(* IEC 61131-3 sources: plcassist-cli/packages/volt-lsp-iec/test-corpus/pro2193/Device/Plc Logic/Application/99 Library/Functions, 16 files *)

(* ---- DWORD_TO_HEXSTRING.fun ---- *)
// Convert PLC memory address into a string with hex characters represented by 0..9 and A..F.
FUNCTION DWORD_TO_HEXSTRING : STRING(8)
VAR_INPUT
	IN		: DWORD;		// Address - result of ADR()
END_VAR
VAR
	i		: USINT;
	temp	: BYTE;
	pt		: POINTER TO BYTE;
END_VAR

(*

Copy from oscat_basic_334 library

version 1.3	29. mar. 2008
programmer	hugo
tested by	tobias

DWORD_TO_STRINGH converts a DWORD to a String of Hexadecimal represented by '0' .. '9' and 'A' .. 'F'.
The lowest order Character will be on the right and the high order Character on the left.

*)

pt	:= ADR(DWORD_TO_HEXSTRING) + 8;					// Read output adress to pointer
pt^	:= 0;											// Write the closing byte (terminator) for the string

FOR i := 1 TO 8 DO									// Write the 8 hex characters backwards
	pt		:= pt - 1;								// Decrement the pointer
	temp	:= TO_BYTE(IN AND 16#0000000F);			// Read the lowest order hex value
	IF temp <= 9 THEN
		pt^	:= enumASCII.NUMBER_0 + temp;			// Convert value to hex character 0 - 9
	ELSE
		pt^	:= enumASCII.UPPERCASE_A + temp - 10;	// Convert value to hex character A - F
	END_IF
	IN		:= SHR(IN, 4);							// Shift 4 bits to right for next hex character
END_FOR

END_FUNCTION

(* ---- GetProjectInfo.fun ---- *)
// Reads the 'application info'. Rightclick on Application, Select Properties, Go to Information tab.
{attribute 'hide_all_locals'}
FUNCTION GetProjectInfo : ProjectInfoType
VAR_INPUT
END_VAR
VAR
	pApp		: POINTER TO CmpApp.APPLICATION;
	pAppInfo	: POINTER TO CmpApp.APPLICATION_INFO;
	iecResult	: SysTypes.RTS_IEC_RESULT;
END_VAR

// Get handle to current PLC application
pApp		:= CmpApp.AppGetCurrent(pResult := ADR(iecResult));
IF pApp = 0 THEN
	GetProjectInfo.projectName	:= 'ERROR READING CURRENT APP';
	RETURN;
END_IF

pAppInfo	:= CmpApp.AppGetApplicationInfo(pApp := pApp, pResult := ADR(iecResult));
IF pAppInfo = 0 THEN
	GetProjectInfo.projectName	:= 'ERROR GETTING APPLICATION INFO';
	RETURN;
END_IF

GetProjectInfo.projectName		:= pAppInfo^.pstProjectName^;
GetProjectInfo.author			:= pAppInfo^.pstAuthor^;
GetProjectInfo.version			:= pAppInfo^.pstVersion^;
GetProjectInfo.description		:= pAppInfo^.pstDescription^;
GetProjectInfo.profile			:= pAppInfo^.pstProfile^;
GetProjectInfo.lastChanges		:= DT_TO_STRING(pAppInfo^.dtLastChanges);

IF GetProjectInfo.projectName = '' THEN
	GetProjectInfo.projectName	:= 'INVALID PROJECTNAME';
END_IF
IF LEN(GetProjectInfo.lastChanges) > 3 THEN
	GetProjectInfo.lastChanges	:= RIGHT(GetProjectInfo.lastChanges, LEN(GetProjectInfo.lastChanges) - 3);
END_IF

END_FUNCTION

(* ---- ParseInstanceName.fun ---- *)
FUNCTION ParseInstanceName
VAR_INPUT
	pInstanceName				: Stu.CharBufferPtr;	// Pointer to string(80)
END_VAR
VAR
	tempString					: STRING(80);
	i							: INT;
END_VAR
VAR CONSTANT
	dotString					: STRING(1) := '.';
	underscoreString			: STRING(1) := '_';
END_VAR

// Check if input string is not empty
IF Stu.StrIsNullOrEmptyA(pInstanceName) THEN
	RETURN;
END_IF

// Check if the input string starts with a known prefix
FOR i := 1 TO 5 DO
	CASE i OF
		1: tempString := 'Device.Application.';
		2: tempString := 'PLC.Application.';
		3: tempString := 'Device.Sim.Device.Application.';
		4: tempString := 'PLC.Sim.PLC.Application.';
		5: tempString := '';
	END_CASE

	IF Stu.StrCmpStartA(pString := pInstanceName, pPrefix := ADR(tempString)) = 0 THEN
		EXIT;
	END_IF
END_FOR

// If prefix is found, remove this prefix
IF i <> 5 THEN
	Stu.StrMidA(
		pst					:= pInstanceName,
		uiInputBufferSize	:= 80,
		iLength				:= TO_INT(StrLenA(pInstanceName) - StrLenA(ADR(tempString))),
		iPosition			:= TO_INT(StrLenA(ADR(tempString)) + 1),
		pstResult			:= pInstanceName,
		uiResultBufferSize	:= 80);
END_IF

// Find all '.' chars and replace with underscores
i := 1;		// Start search at position 1
WHILE (i := StrFindA(pst1 := pInstanceName, pst2 := ADR(dotString), uiSearchStart := TO_UINT(i))) > 0 DO
	StrReplaceA(
		pstInput			:= pInstanceName,
		uiInputBufferSize	:= 80,
		pstReplaceWith		:= ADR(underscoreString),
		iLengthInput		:= 1,	// Don't know function of this parameter..
		iLengthToReplace	:= 1,
		iLengthToReplaceWith:= 1,
		iPosition			:= i);	// i is position where the dot was found
END_WHILE

END_FUNCTION

(* ---- RANGE_TO_RANGE.fun ---- *)
// Used for mapping a real input value from one range to another.
FUNCTION RANGE_TO_RANGE : REAL
VAR_INPUT
	input		: REAL;	// input is limited to: input_LO <= input <= input_HI
	input_LO	: REAL;
	input_HI	: REAL;
	output_LO	: REAL;
	output_HI	: REAL;
END_VAR
VAR
	inputRange	: REAL;
	outputRange	: REAL;
END_VAR

(*

Zie hier voor voorbeeld:
https://stackoverflow.com/questions/929103/convert-a-number-range-to-another-range-maintaining-ratio

Update 24-03-2023: Added logic from SCALE_R function in Oscat library.
*)

inputRange	:= input_HI - input_LO;
outputRange	:= output_HI - output_LO;

IF inputRange = 0 THEN // Never divide by zero
	RANGE_TO_RANGE := output_LO;
ELSE
	RANGE_TO_RANGE := outputRange / inputRange * (LIMIT(input_LO, input, input_HI) - input_LO) + output_LO;
END_IF

END_FUNCTION

(* ---- RANGE_TO_WORD.fun ---- *)
// Used for mapping a REAL input value into a WORD (from 0 to 65535)
FUNCTION RANGE_TO_WORD : WORD
VAR_INPUT
	input		: REAL;	// input is limited to: input_LO <= input <= input_HI
	input_LO	: REAL;
	input_HI	: REAL;
END_VAR

// Update 24-03-2023: Added logic from RANGE_TO_WORD function in Oscat library.
// Update 08-06-2023: Removed logic here and use RANGE_TO_RANGE method instead (because devide by zero exception was possible)

RANGE_TO_WORD := TO_WORD(
					TRUNC(
						RANGE_TO_RANGE(
							input		:= input,
							input_LO	:= input_LO,
							input_HI	:= input_HI,
							output_LO	:= 0.0,
//							output_HI	:= 65535.0)));
							output_HI	:= 16384.0)));		// For Lenze analog outputs the maximum range is 16384.

// Example use:
// MapAnalogOut			:= Brink.RANGE_TO_WORD(input := rSetPointCharger,			input_LO := 0.0,	input_HI := rMaxChargerSetting);
// MapAnalogOut			:= Brink.RANGE_TO_WORD(input := profile.rVel,				input_LO := 0.0,	input_HI := rMaxSpeedSetting);
// wSetPointCharger		:= Brink.RANGE_TO_WORD(input := Data.rSetPointCharger,		input_LO := 0.0,	input_HI := 20.0);
// wSetPointCharger[i]	:= Brink.RANGE_TO_WORD(input := Data.rSetPointCharger[i],	input_LO := 0.0,	input_HI := 20.0);

END_FUNCTION

(* ---- Round.fun ---- *)
// This function rounds a real down to n digits behind the comma.
FUNCTION Round : REAL
VAR_INPUT
	in	: REAL;
	N	: USINT(0..4);
END_VAR
VAR
	X	: REAL;
END_VAR

(*
version 1.5	25. oct. 2008
programmer	hugo
tested by	tobias

this function rounds a real down to n digits behind the comma.

*)

CASE N OF
	0:	X := 1.0;
	1:	X := 10.0;
	2:	X := 100.0;
	3:	X := 1000.0;
	4:	X := 10000.0;
END_CASE

Round := TO_REAL(TO_DINT(in * X)) / X;

(* revision history
hm	1. sep 2006	rev 1.0
	original version

hm	2. dec 2007	rev 1.1
	changed code for better performance

hm	8. jan 2008	rev 1.2
	further improvement in performance

hm 11. mar. 2008	rev 1.3
	corrected an error with negative numbers
	use real_to_dint instead of trunc

hm	16. mar 2008	rev 1.4
	added type conversion to avoid warning under codesys 3.0

hm	25. oct. 2008	rev 1.5
	new code using global constants decades
*)

END_FUNCTION

(* ---- TaskDisableWatchdog.fun ---- *)
// Disable watchdog for the current task
// The watchdog is disabled only for the current cycle! At the next cycle, the watchod is automatically enabled!
FUNCTION TaskDisableWatchdog : BOOL
VAR
	iecResult		: SysTypes.RTS_IEC_RESULT;
	handle			: SysTypes.RTS_IEC_HANDLE;
END_VAR

handle				:= CmpIecTask.IecTaskGetCurrent(ADR(iecResult));			// Function to get own task handle

IF handle = SysTypes.RTS_INVALID_HANDLE THEN RETURN; END_IF
IF iecResult <> CmpErrors.Errors.ERR_OK THEN RETURN; END_IF

iecResult			:= CmpIecTask.IecTaskDisableWatchdog(hIecTask := handle);

IF iecResult <> CmpErrors.Errors.ERR_OK THEN RETURN; END_IF

TaskDisableWatchdog	:= TRUE;

END_FUNCTION

(* ---- TaskGetInfo.fun ---- *)
// Returns task interval value (in ms) of current task
// Do not call function each PLC cycle. Calling it once is enough.
FUNCTION TaskGetInfo : CmpIecTask.Task_Info2
VAR
	iecResult		: SysTypes.RTS_IEC_RESULT;
	handle			: SysTypes.RTS_IEC_HANDLE;
	pIecTaskInfo	: POINTER TO CmpIecTask.Task_Info2;
END_VAR

handle				:= CmpIecTask.IecTaskGetCurrent(ADR(iecResult));			// Function to get own task handle

IF handle = SysTypes.RTS_INVALID_HANDLE THEN RETURN; END_IF
IF iecResult <> CmpErrors.Errors.ERR_OK THEN RETURN; END_IF

pIecTaskInfo		:= CmpIecTask.IecTaskGetInfo3(hIecTask := handle, pResult := ADR(iecResult));	// Function returns the task information of the specified task

IF pIecTaskInfo = 0 THEN RETURN; END_IF

TaskGetInfo			:= pIecTaskInfo^;

END_FUNCTION

(* ---- TaskGetInterval.fun ---- *)
// Returns task interval value (in ms) of current task
// Do not call function each PLC cycle. Calling it once is enough.
FUNCTION TaskGetInterval : TIME
VAR_OUTPUT
	taskName		: STRING;
END_VAR
VAR
	iecResult		: SysTypes.RTS_IEC_RESULT;
	handle			: SysTypes.RTS_IEC_HANDLE;
	pIecTaskInfo	: POINTER TO CmpIecTask.Task_Info2;
END_VAR

handle				:= CmpIecTask.IecTaskGetCurrent(ADR(iecResult));			// Function to get own task handle

IF handle = SysTypes.RTS_INVALID_HANDLE THEN RETURN; END_IF
IF iecResult <> CmpErrors.Errors.ERR_OK THEN RETURN; END_IF

pIecTaskInfo		:= CmpIecTask.IecTaskGetInfo3(hIecTask := handle, pResult := ADR(iecResult));	// Function returns the task information of the specified task

IF pIecTaskInfo = 0 THEN RETURN; END_IF

taskName			:= pIecTaskInfo^.pszName^;
TaskGetInterval		:= TO_TIME(pIecTaskInfo^.dwInterval / 1000);

END_FUNCTION

(* ---- ThrowException.fun ---- *)
FUNCTION ThrowException : BOOL
VAR_INPUT
	message			: STRING := '';	// A custom message (reason of throwing the exception) to echo to the PLC log
END_VAR

LogPlc.Fatal(message);		// Add a custom message to the PLC log
LogPlc.Throw();

END_FUNCTION

(* ---- Arrays.prg ---- *)
// Helper functions for arrays
{attribute 'no_explicit_call' := 'Static helper class to do stuff with all kinds of arrays'}
{attribute 'hide_all_locals'}
PROGRAM Arrays

// Because arrays are value-type, it's not possible to cast an array of fbs to another type.
// More info here:
// https://stackoverflow.com/questions/69319659/how-do-i-pass-an-array-of-an-extended-type-in-codesys-twincat3

// The function Vacuum_ResetAll should not be needed !!!
// The interface IVacuum extends IActuator,
// so you should be able to use ActuatorResetAll for vacuums too
// However, this does not work with dynamic arrays
// You get error message: Cannot convert type 'ARRAY[1..3] of IVacuum' to type 'ARRAY[*] of IActuator
// Hopefully CODESYS fixes this in the future.

END_PROGRAM

// Returns true if all elements in the actuator array are equal to condition.
METHOD PUBLIC Actuator_All : BOOL
VAR_IN_OUT
	actuatorArray		: ARRAY[*] OF IActuator;
END_VAR
VAR_INPUT
	condition			: BOOL;
END_VAR
VAR
	upper, lower, di	: DINT;
END_VAR
%FOLDER Tests
lower	:= LOWER_BOUND(actuatorArray, 1);
upper	:= UPPER_BOUND(actuatorArray, 1);

Actuator_All := TRUE;

FOR di := lower TO upper DO
	IF actuatorArray[di] = 0 THEN
		LogPlc.Fatal('Actuator_All: Element in array of interfaces is NULL!');
		Actuator_All := FALSE;
		EXIT;
	ELSIF actuatorArray[di].Map() <> condition THEN
		Actuator_All := FALSE;
		EXIT;	// Exit the loop on the first match
	END_IF
END_FOR
END_METHOD

// Returns true if any element in the actuator array is equal to condition.
METHOD PUBLIC Actuator_Any : BOOL
VAR_IN_OUT
	actuatorArray		: ARRAY[*] OF IActuator;
END_VAR
VAR_INPUT
	condition			: BOOL;
END_VAR
VAR
	upper, lower, di	: DINT;
END_VAR
%FOLDER Tests
lower	:= LOWER_BOUND(actuatorArray, 1);
upper	:= UPPER_BOUND(actuatorArray, 1);

FOR di := lower TO upper DO
	IF actuatorArray[di] = 0 THEN
		LogPlc.Fatal('Actuator_Any: Element in array of interfaces is NULL!');
	ELSIF actuatorArray[di].Map() = condition THEN
		Actuator_Any := TRUE;
		EXIT;	// Exit the loop on the first match
	END_IF
END_FOR
END_METHOD

// Fires the Reset method on the actuator array
METHOD PUBLIC Actuator_ResetAll
VAR_IN_OUT
	actuatorArray		: ARRAY[*] OF IActuator;
END_VAR
VAR
	upper, lower, di	: DINT;
END_VAR
%FOLDER Execute methods
lower	:= LOWER_BOUND(actuatorArray, 1);
upper	:= UPPER_BOUND(actuatorArray, 1);

FOR di := lower TO upper DO
	IF actuatorArray[di] = 0 THEN
		LogPlc.Fatal('Actuator_ResetAll: Element in array of interfaces is NULL!');
	ELSE
		actuatorArray[di].Reset();
	END_IF
END_FOR
END_METHOD

// Returns true if all the modules (Xi, Xu, or Y unit) are in a safe position
METHOD PUBLIC AllUnitsAreInSafePosition : BOOL
VAR_IN_OUT
	safeModules			: ARRAY[*] OF IModuleHasSafePos;
END_VAR
VAR
	upper, lower, di	: DINT;
END_VAR
%FOLDER Tests
lower	:= LOWER_BOUND(safeModules, 1);
upper	:= UPPER_BOUND(safeModules, 1);

AllUnitsAreInSafePosition := TRUE;

FOR di := lower TO upper DO
	IF safeModules[di] = 0 THEN
		ThrowException('AllUnitsAreInSafePosition: Element in array of interfaces is NULL!');
	ELSIF NOT safeModules[di].InSafePos THEN
		AllUnitsAreInSafePosition := FALSE;
		EXIT;	// Exit the loop on the first match
	END_IF
END_FOR
END_METHOD

// Returns true if all elements in the bool array are equal to condition
METHOD PUBLIC Bool_All : BOOL
VAR_IN_OUT
	boolArray			: ARRAY[*] OF BOOL;
END_VAR
VAR_INPUT
	condition			: BOOL;
END_VAR
VAR
	upper, lower, di	: DINT;
END_VAR
%FOLDER Tests
lower	:= LOWER_BOUND(boolArray, 1);
upper	:= UPPER_BOUND(boolArray, 1);

Bool_All := TRUE;

FOR di := lower TO upper DO
	IF boolArray[di] <> condition THEN
		Bool_All := FALSE;
		EXIT;						// Exit the loop on the first match
	END_IF
END_FOR
END_METHOD

// Returns true if any element in the bool array is equal to condition
METHOD PUBLIC Bool_Any : BOOL
VAR_IN_OUT
	boolArray			: ARRAY[*] OF BOOL;
END_VAR
VAR_INPUT
	condition			: BOOL;
END_VAR
VAR
	upper, lower, di	: DINT;
END_VAR
%FOLDER Tests
lower	:= LOWER_BOUND(boolArray, 1);
upper	:= UPPER_BOUND(boolArray, 1);

FOR di := lower TO upper DO
	IF boolArray[di] = condition THEN
		Bool_Any := TRUE;
		EXIT;						// Exit the loop on the first match
	END_IF
END_FOR
END_METHOD

// Resets all booleans in an array
METHOD PUBLIC Bool_Reset
VAR_IN_OUT
	boolArray		: ARRAY[*] OF BOOL;
END_VAR
VAR
	upper, lower, di	: DINT;
END_VAR
%FOLDER Execute methods
lower	:= LOWER_BOUND(boolArray, 1);
upper	:= UPPER_BOUND(boolArray, 1);

FOR di := lower TO upper DO
	boolArray[di] := FALSE;
END_FOR
END_METHOD

// Sets all booleans in an array
METHOD PUBLIC Bool_Set
VAR_IN_OUT
	boolArray		: ARRAY[*] OF BOOL;
END_VAR
VAR
	upper, lower, di	: DINT;
END_VAR
%FOLDER Execute methods
lower	:= LOWER_BOUND(boolArray, 1);
upper	:= UPPER_BOUND(boolArray, 1);

FOR di := lower TO upper DO
	boolArray[di] := TRUE;
END_FOR
END_METHOD

// Returns true if all digital sensors in the array are equal to condition
METHOD PUBLIC DigitalSensor_All : BOOL
VAR_IN_OUT
	sensorArray			: ARRAY[*] OF DigitalSensorFB;
END_VAR
VAR_INPUT
	condition			: BOOL;		// TRUE = IsActive, FALSE = IsInactive
END_VAR
VAR
	upper, lower, di	: DINT;
END_VAR
%FOLDER Digital Sensors
lower	:= LOWER_BOUND(sensorArray, 1);
upper	:= UPPER_BOUND(sensorArray, 1);

DigitalSensor_All := TRUE;

FOR di := lower TO upper DO
	IF (condition AND NOT sensorArray[di].IsActive)
	OR (NOT condition AND NOT sensorArray[di].IsInactive)
	THEN
		DigitalSensor_All := FALSE;
		EXIT;						// Exit the loop on the first match
	END_IF
END_FOR
END_METHOD

// Returns true if any element in the bool array is equal to condition
METHOD PUBLIC DigitalSensor_Any : BOOL
VAR_IN_OUT
	sensorArray			: ARRAY[*] OF DigitalSensorFB;
END_VAR
VAR_INPUT
	condition			: BOOL;
END_VAR
VAR
	upper, lower, di	: DINT;
END_VAR
%FOLDER Digital Sensors
lower	:= LOWER_BOUND(sensorArray, 1);
upper	:= UPPER_BOUND(sensorArray, 1);

FOR di := lower TO upper DO
	IF (condition AND sensorArray[di].IsActive)
	OR (NOT condition AND sensorArray[di].IsInactive)
	THEN
		DigitalSensor_Any := TRUE;
		EXIT;						// Exit the loop on the first match
	END_IF
END_FOR
END_METHOD

// Returns true if all digital sensors (that are enabled) in the array are equal to condition
METHOD PUBLIC DigitalSensor_Enabled_All : BOOL
VAR_IN_OUT
	sensorArray			: ARRAY[*] OF DigitalSensorWithEnableFB;
END_VAR
VAR_INPUT
	bitMask				: DWORD;	// Only test sensors when corresponding bitnumber is high.
	condition			: BOOL;
END_VAR
VAR
	upper, lower, di	: DINT;
	counter				: USINT := 0;
END_VAR
%FOLDER Digital Sensors
lower	:= LOWER_BOUND(sensorArray, 1);
upper	:= UPPER_BOUND(sensorArray, 1);

DigitalSensor_Enabled_All := TRUE;

FOR di := lower TO upper DO

	IF NOT BitLogic.Extract(bitMask, counter) THEN	// not cavity disabled
		IF (condition AND NOT sensorArray[di].IsActive)
		OR (NOT condition AND NOT sensorArray[di].IsInactive)
		THEN
			IF sensorArray[di].IsEnabled THEN		//Only reset when sensor is enabled
				DigitalSensor_Enabled_All := FALSE;
				EXIT;						// Exit the loop on the first match
			END_IF
		END_IF
	END_IF

	Increment.AnyInt(counter);
END_FOR
END_METHOD

// Returns true if any element (that is enabled) in the bool array is equal to condition
METHOD PUBLIC DigitalSensor_Enabled_Any : BOOL
VAR_IN_OUT
	sensorArray			: ARRAY[*] OF DigitalSensorWithEnableFB;
END_VAR
VAR_INPUT
	bitMask				: DWORD;	// Only test sensors when corresponding bitnumber is high.
	condition			: BOOL;
END_VAR
VAR
	upper, lower, di	: DINT;
	counter				: USINT := 0;
END_VAR
%FOLDER Digital Sensors
lower	:= LOWER_BOUND(sensorArray, 1);
upper	:= UPPER_BOUND(sensorArray, 1);

FOR di := lower TO upper DO

	IF NOT BitLogic.Extract(bitMask, counter) THEN	// not cavity disabled
		IF (condition AND sensorArray[di].IsActive)
		OR (NOT condition AND sensorArray[di].IsInactive)
		THEN
			IF sensorArray[di].IsEnabled THEN		// Only set when sensor is enabled
				DigitalSensor_Enabled_Any := TRUE;
				EXIT;						// Exit the loop on the first match
			END_IF
		END_IF
	END_IF

	Increment.AnyInt(counter);
END_FOR
END_METHOD

// Returns the largest position in an array
METHOD PUBLIC Position_Largest : REAL
VAR_IN_OUT
	positionArray		: ARRAY[*] OF PositionWithProfileType;
END_VAR
VAR
	upper, lower, di	: DINT;
END_VAR
%FOLDER Positions
lower					:= LOWER_BOUND(positionArray, 1);
upper					:= UPPER_BOUND(positionArray, 1);
Position_Largest		:= GVL_Constants.RealSmallest;

FOR di := lower TO upper DO
	Position_Largest	:= MAX(positionArray[di].Pos.value, Position_Largest);
END_FOR
END_METHOD

// Returns the smallest position in an array
METHOD PUBLIC Position_Smallest : REAL
VAR_IN_OUT
	positionArray		: ARRAY[*] OF PositionWithProfileType;
END_VAR
VAR
	upper, lower, di	: DINT;
END_VAR
%FOLDER Positions
lower					:= LOWER_BOUND(positionArray, 1);
upper					:= UPPER_BOUND(positionArray, 1);
Position_Smallest		:= GVL_Constants.RealLargest;

FOR di := lower TO upper DO
	Position_Smallest	:= MIN(positionArray[di].Pos.value, Position_Smallest);
END_FOR
END_METHOD

// Returns true if all elements in the vacuum array are equal to condition. Option to test either vacuum high input, or vacuum set output.
METHOD PUBLIC Vacuum_All : BOOL
VAR_IN_OUT
	vacuumArray			: ARRAY[*] OF IVacuum;
END_VAR
VAR_INPUT
	condition			: BOOL;
	channel				: enumSelectIQ := enumSelectIQ.Output;	// Optional: Select to check the vacuum high input, the set output, or both
END_VAR
VAR
	upper, lower, di	: DINT;
END_VAR
%FOLDER Tests
lower	:= LOWER_BOUND(vacuumArray, 1);
upper	:= UPPER_BOUND(vacuumArray, 1);

Vacuum_All := TRUE;

FOR di := lower TO upper DO
	IF vacuumArray[di] = 0 THEN
		LogPlc.Fatal('Vacuum_All: Element in array of interfaces is NULL!');
		Vacuum_All := FALSE;
		EXIT;	// Exit the loop on the first match
	END_IF

	IF vacuumArray[di].IsHigh <> condition AND (channel = enumSelectIQ.Input OR channel = enumSelectIQ.Both)
	OR vacuumArray[di].IsTurnedOn <> condition AND (channel = enumSelectIQ.Output OR channel = enumSelectIQ.Both)
	THEN
		Vacuum_All := FALSE;
		EXIT;	// Exit the loop on the first match
	END_IF
END_FOR
END_METHOD

// Returns true if any element in the vacuum array is equal to condition. Option to test either vacuum high input, or vacuum set output.
METHOD PUBLIC Vacuum_Any : BOOL
VAR_IN_OUT
	vacuumArray			: ARRAY[*] OF IVacuum;
END_VAR
VAR_INPUT
	condition			: BOOL;
	channel				: enumSelectIQ := enumSelectIQ.Output;	// Optional: Select to check the vacuum high input, the set output, or both
END_VAR
VAR
	upper, lower, di	: DINT;
END_VAR
%FOLDER Tests
lower	:= LOWER_BOUND(vacuumArray, 1);
upper	:= UPPER_BOUND(vacuumArray, 1);

FOR di := lower TO upper DO
	IF vacuumArray[di] = 0 THEN
		LogPlc.Fatal('Vacuum_Any: Element in array of interfaces is NULL!');
		CONTINUE;
	END_IF
	CASE channel OF
		enumSelectIQ.Input:
			IF vacuumArray[di].IsHigh = condition THEN
				Vacuum_Any := TRUE;
				EXIT;	// Exit the loop on the first match
			END_IF
		enumSelectIQ.Output:
			IF vacuumArray[di].IsTurnedOn = condition THEN
				Vacuum_Any := TRUE;
				EXIT;	// Exit the loop on the first match
			END_IF
		enumSelectIQ.Both:
			IF vacuumArray[di].IsHigh = condition OR vacuumArray[di].IsTurnedOn = condition THEN
				Vacuum_Any := TRUE;
				EXIT;	// Exit the loop on the first match
			END_IF
	END_CASE
END_FOR
END_METHOD

// Returns true if all elements in the vacuum array (that are enabled) are equal to condition. Option to test either vacuum high input, or vacuum set output.
METHOD PUBLIC Vacuum_Enabled_All : BOOL
VAR_IN_OUT
	vacuumArray			: ARRAY[*] OF IVacuum;
END_VAR
VAR_INPUT
	bitMask				: WORD;	// Only test vacuums when corresponding bitnumber is high.
	condition			: BOOL;
	channel				: enumSelectIQ := enumSelectIQ.Output;	// Optional: Select to check the vacuum high input, the set output, or both
END_VAR
VAR
	upper, lower, di	: DINT;
END_VAR
%FOLDER Tests
lower	:= LOWER_BOUND(vacuumArray, 1);
upper	:= UPPER_BOUND(vacuumArray, 1);

Vacuum_Enabled_All := TRUE;

FOR di := lower TO upper DO
	IF vacuumArray[di] = 0 THEN
		LogPlc.Fatal('Vacuum_All: Element in array of interfaces is NULL!');
		Vacuum_Enabled_All := FALSE;
		EXIT;	// Exit the loop on the first match
	END_IF

	IF NOT BitLogic.Extract(bitMask, TO_USINT(di)) THEN
		CONTINUE;
	END_IF

	IF vacuumArray[di].IsHigh <> condition AND (channel = enumSelectIQ.Input OR channel = enumSelectIQ.Both)
	OR vacuumArray[di].IsTurnedOn <> condition AND (channel = enumSelectIQ.Output OR channel = enumSelectIQ.Both)
	THEN
		Vacuum_Enabled_All := FALSE;
		EXIT;	// Exit the loop on the first match
	END_IF
END_FOR
END_METHOD

// Returns true if any element in the vacuum array (that is enabled) is equal to condition. Option to test either vacuum high input, or vacuum set output.
METHOD PUBLIC Vacuum_Enabled_Any : BOOL
VAR_IN_OUT
	vacuumArray			: ARRAY[*] OF IVacuum;
END_VAR
VAR_INPUT
	bitMask				: WORD;	// Only test vacuums when corresponding bitnumber is high.
	condition			: BOOL;
	channel				: enumSelectIQ := enumSelectIQ.Output;	// Optional: Select to check the vacuum high input, the set output, or both
END_VAR
VAR
	upper, lower, di	: DINT;
END_VAR
%FOLDER Tests
lower	:= LOWER_BOUND(vacuumArray, 1);
upper	:= UPPER_BOUND(vacuumArray, 1);

FOR di := lower TO upper DO
	IF vacuumArray[di] = 0 THEN
		LogPlc.Fatal('Vacuum_Any: Element in array of interfaces is NULL!');
		CONTINUE;
	END_IF

	IF NOT BitLogic.Extract(bitMask, TO_USINT(di)) THEN
		CONTINUE;
	END_IF

	CASE channel OF
		enumSelectIQ.Input:
			IF vacuumArray[di].IsHigh = condition THEN
				Vacuum_Enabled_Any := TRUE;
				EXIT;	// Exit the loop on the first match
			END_IF
		enumSelectIQ.Output:
			IF vacuumArray[di].IsTurnedOn = condition THEN
				Vacuum_Enabled_Any := TRUE;
				EXIT;	// Exit the loop on the first match
			END_IF
		enumSelectIQ.Both:
			IF vacuumArray[di].IsHigh = condition OR vacuumArray[di].IsTurnedOn = condition THEN
				Vacuum_Enabled_Any := TRUE;
				EXIT;	// Exit the loop on the first match
			END_IF
	END_CASE
END_FOR
END_METHOD

// Fires the Release method on all elements in the vacuum array
METHOD PUBLIC Vacuum_ReleaseAll : BOOL
VAR_IN_OUT
	vacuumArray			: ARRAY[*] OF IVacuum;
END_VAR
VAR
	upper, lower, di	: DINT;
END_VAR
%FOLDER Execute methods
lower	:= LOWER_BOUND(vacuumArray, 1);
upper	:= UPPER_BOUND(vacuumArray, 1);

Vacuum_ReleaseAll := TRUE;

FOR di := lower TO upper DO
	IF vacuumArray[di] = 0 THEN
		LogPlc.Fatal('Vacuum_ReleaseAll: Element in array of interfaces is NULL!');
		Vacuum_ReleaseAll := FALSE;
	ELSIF NOT vacuumArray[di].Release() THEN
		Vacuum_ReleaseAll := FALSE;
	END_IF
END_FOR
END_METHOD

// Fires the Release method on some elements in the vacuum array. Only reset vacuums whose corresponding bit is high in the bitMask
// !Remember! Vacuum arrays usually start from 1. So to set the first vacuum, use the second bit (bitMask.1) in the bitMask!
METHOD PUBLIC Vacuum_ReleaseSelected : BOOL
VAR_IN_OUT
	vacuumArray			: ARRAY[*] OF IVacuum;
END_VAR
VAR_INPUT
	bitMask				: WORD;	// Release vacuum if corresponding bitnumber is high.
END_VAR
VAR
	upper, lower, di	: DINT;
END_VAR
%FOLDER Execute methods
lower	:= LOWER_BOUND(vacuumArray, 1);
upper	:= UPPER_BOUND(vacuumArray, 1);

Vacuum_ReleaseSelected := TRUE;

FOR di := lower TO upper DO
	IF BitLogic.Extract(bitMask, TO_USINT(di)) THEN
		IF vacuumArray[di] = 0 THEN
			LogPlc.Fatal('Vacuum_ReleaseSelected: Element in array of interfaces is NULL!');
			Vacuum_ReleaseSelected := FALSE;
		ELSIF NOT vacuumArray[di].Release() THEN
			Vacuum_ReleaseSelected := FALSE;
		END_IF
	END_IF
END_FOR

// Method will fail if upper limit of vacuum array > 16
END_METHOD

// Resets the vacuum suction cups that no longer have a product. Returns 0 if all suction cups are turned off.
METHOD PUBLIC Vacuum_ResetIfNotHigh : UINT
VAR_IN_OUT
	vacuumArray			: ARRAY[*] OF IVacuum;
END_VAR
VAR
	result				: UINT;
	upper, lower, di	: DINT;
END_VAR
%FOLDER Execute methods
lower	:= LOWER_BOUND(vacuumArray, 1);
upper	:= UPPER_BOUND(vacuumArray, 1);

FOR di := lower TO upper DO
	IF vacuumArray[di] = 0 THEN
		LogPlc.Fatal('Vacuum_ResetIfNotHigh: Element in array of interfaces is NULL!');
	ELSIF vacuumArray[di].IsHigh THEN
		BitLogic.Load(result, TRUE, TO_USINT(LIMIT(0, di, 15)));
	ELSE
		vacuumArray[di].Reset();
	END_IF
END_FOR

Vacuum_ResetIfNotHigh := result;
END_METHOD

// Returns true if some elements in the vacuum array are equal to condition.
// Only test vacuums whose corresponding bit is high in the bitMask
// Option to test either vacuum high input, or vacuum set output.
// !Remember! Vacuum arrays usually start from 1. So to set the first vacuum, use the second bit (bitMask.1) in the bitMask!
METHOD PUBLIC Vacuum_Selected : BOOL
VAR_IN_OUT
	vacuumArray			: ARRAY[*] OF IVacuum;
END_VAR
VAR_INPUT
	bitMask				: WORD;	// Test vacuum if corresponding bitnumber is high.
	condition			: BOOL;
	channel				: enumSelectIQ := enumSelectIQ.Output;	// Optional: Select to check the vacuum high input, the set output, or both
END_VAR
VAR
	upper, lower, di	: DINT;
END_VAR
%FOLDER Tests
lower	:= LOWER_BOUND(vacuumArray, 1);
upper	:= UPPER_BOUND(vacuumArray, 1);

Vacuum_Selected := TRUE;

FOR di := lower TO upper DO
	IF BitLogic.Extract(bitMask, TO_USINT(di)) THEN
		IF vacuumArray[di] = 0 THEN
			LogPlc.Fatal('Vacuum_Selected: Element in array of interfaces is NULL!');
			Vacuum_Selected := FALSE;
			EXIT;
		END_IF
		CASE channel OF
			enumSelectIQ.Input:
				IF vacuumArray[di].IsHigh <> condition THEN
					Vacuum_Selected := FALSE;
					EXIT;	// Exit the loop on the first match
				END_IF
			enumSelectIQ.Output:
				IF vacuumArray[di].IsTurnedOn <> condition THEN
					Vacuum_Selected := FALSE;
					EXIT;	// Exit the loop on the first match
				END_IF
			enumSelectIQ.Both:
				IF vacuumArray[di].IsHigh <> condition OR vacuumArray[di].IsTurnedOn <> condition THEN
					Vacuum_Selected := FALSE;
					EXIT;	// Exit the loop on the first match
				END_IF
		END_CASE
	END_IF
END_FOR

// Method will fail if upper limit of vacuum array > 16
END_METHOD

// Fires the Set method on all elements in the vacuum array. Return true if all vacuums are high.
METHOD PUBLIC Vacuum_SetAll : BOOL
VAR_IN_OUT
	vacuumArray			: ARRAY[*] OF IVacuum;
END_VAR
VAR
	upper, lower, di	: DINT;
END_VAR
%FOLDER Execute methods
lower	:= LOWER_BOUND(vacuumArray, 1);
upper	:= UPPER_BOUND(vacuumArray, 1);

Vacuum_SetAll := TRUE;

FOR di := lower TO upper DO
	IF vacuumArray[di] = 0 THEN
		LogPlc.Fatal('Vacuum_SetAll: Element in array of interfaces is NULL!');
		Vacuum_SetAll := FALSE;
	ELSIF NOT vacuumArray[di].Set() THEN
		Vacuum_SetAll := FALSE;
	END_IF
END_FOR
END_METHOD

// Fires the Set method on some elements in the vacuum array. Only set vacuums whose corresponding bit is high in the bitMask
// !Remember! Vacuum arrays usually start from 1. So to set the first vacuum, use the second bit (bitMask.1) in the bitMask!
METHOD PUBLIC Vacuum_SetSelected : BOOL
VAR_IN_OUT
	vacuumArray			: ARRAY[*] OF IVacuum;
END_VAR
VAR_INPUT
	bitMask				: WORD;	// Set vacuum if corresponding bitnumber is high.
END_VAR
VAR
	upper, lower, di	: DINT;
END_VAR
%FOLDER Execute methods
lower	:= LOWER_BOUND(vacuumArray, 1);
upper	:= UPPER_BOUND(vacuumArray, 1);

Vacuum_SetSelected := TRUE;

FOR di := lower TO upper DO
	IF BitLogic.Extract(bitMask, TO_USINT(di)) THEN
		IF vacuumArray[di] = 0 THEN
			LogPlc.Fatal('Vacuum_SetSelected: Element in array of interfaces is NULL!');
			Vacuum_SetSelected := FALSE;
		ELSIF NOT vacuumArray[di].Set() THEN
			Vacuum_SetSelected := FALSE;
		END_IF
	END_IF
END_FOR

// Method will fail if upper limit of vacuum array > 16
END_METHOD

(* ---- BitLogic.prg ---- *)
// Helper functions to set or reset bits in integers
{attribute 'no_explicit_call' := 'Static helper class to do various operations on bits in integers'}
{attribute 'hide_all_locals'}
PROGRAM BitLogic
VAR
	uInput		: PointerSizesUnion;
END_VAR

END_PROGRAM

// Population count: Count the number of bits that are 1 in a byte
METHOD PUBLIC CountByte : USINT
VAR_INPUT
	in	: BYTE;			// Count number of 1's
END_VAR

// This method uses Brian Kernighan's algorithm. Google it for more info.
WHILE in <> 0 DO
	in			:= in AND (in - 1);		// Subtracting 1 from a number flips all the bits after the rightmost set bit, including the rightmost set bit itself
	CountByte	:= CountByte + 1;
END_WHILE
END_METHOD

// Population count: Count the number of bits that are 1 in a dword
METHOD PUBLIC CountDWord : USINT
VAR_INPUT
	in	: DWORD;		// Count number of 1's
END_VAR

// This method uses Brian Kernighan's algorithm. Google it for more info.
WHILE in <> 0 DO
	in			:= in AND (in - 1);
	CountDWord	:= CountDWord + 1;
END_WHILE
END_METHOD

// Population count: Count the number of bits that are 1 in a word
METHOD PUBLIC CountWord : USINT
VAR_INPUT
	in	: WORD;			// Count number of 1's
END_VAR

// This method uses Brian Kernighan's algorithm. Google it for more info.
WHILE in <> 0 DO
	in			:= in AND (in - 1);
	CountWord	:= CountWord + 1;
END_WHILE
END_METHOD

// Extract a single bit from any integer type (usefull in FOR loops)
METHOD PUBLIC Extract : BOOL
VAR_INPUT
	in	: ANY_INT;		// extract bit from this integer
	N	: USINT(0..63);	// position of bit on the nth position from right (right is lowest bit)
END_VAR
ValidateInput(in.diSize, N);

uInput.p1_Byte := in.pValue;

CASE in.diSize OF
	1:	Extract := (SHR(uInput.p1_Byte^,	N) AND 16#00000001) > 0;
	2:	Extract := (SHR(uInput.p2_Word^,	N) AND 16#00000001) > 0;
	4:	Extract := (SHR(uInput.p4_DWord^,	N) AND 16#00000001) > 0;
	8:	Extract := (SHR(uInput.p8_LWord^,	N) AND 16#00000001) > 0;
END_CASE
END_METHOD

// Extract a single bit from a byte type (usefull in FOR loops)
METHOD PUBLIC ExtractFromByte : BOOL
VAR_INPUT
	in	: REFERENCE TO BYTE;	// extract bit from this byte
	N	: BYTE(0..7);			// position of bit on the nth position from right (right is lowest bit)
END_VAR

// This is a separate method from Extract(), because ANY_INT cannot be a reference.
ExtractFromByte := (SHR(in,	N) AND 16#00000001) > 0;
END_METHOD

// Extract a single bit from a DWORD type (usefull in FOR loops)
METHOD PUBLIC ExtractFromDWord : BOOL
VAR_INPUT
	in	: REFERENCE TO DWORD;	// extract bit from this byte
	N	: BYTE(0..31);			// position of bit on the nth position from right (right is lowest bit)
END_VAR

// This is a separate method from Extract(), because ANY_INT cannot be a reference.
ExtractFromDWord := (SHR(in, N) AND 16#00000000_00000000_00000000_00000001) > 0;
END_METHOD

// Extract a single bit from a WORD type (usefull in FOR loops)
METHOD PUBLIC ExtractFromWord : BOOL
VAR_INPUT
	in	: REFERENCE TO WORD;	// extract bit from this byte
	N	: BYTE(0..15);			// position of bit on the nth position from right (right is lowest bit)
END_VAR

// This is a separate method from Extract(), because ANY_INT cannot be a reference.
ExtractFromWord := (SHR(in, N) AND 16#00000000_00000001) > 0;
END_METHOD

// Load a bit into any integer at position N
METHOD PUBLIC Load
VAR_INPUT
	in	: ANY_INT;		// Set or reset a bit in this integer
	val	: BOOL;			// The value to set
	N	: USINT(0..63);	// position of bit on the nth position from right (right is lowest bit)
END_VAR
ValidateInput(in.diSize, N);

uInput.p1_Byte := in.pValue;

CASE in.diSize OF
	1:	uInput.p1_Byte^		:= SEL(val, uInput.p1_Byte^  AND (NOT SHL( BYTE#1, N)),	uInput.p1_Byte^  OR SHL( BYTE#1, N));
	2:	uInput.p2_Word^		:= SEL(val, uInput.p2_Word^	 AND (NOT SHL( WORD#1, N)),	uInput.p2_Word^  OR SHL( WORD#1, N));
	4:	uInput.p4_DWord^	:= SEL(val, uInput.p4_DWord^ AND (NOT SHL(DWORD#1, N)),	uInput.p4_DWord^ OR SHL(DWORD#1, N));
	8:	uInput.p8_LWord^	:= SEL(val, uInput.p8_LWord^ AND (NOT SHL(LWORD#1, N)),	uInput.p8_LWord^ OR SHL(LWORD#1, N));
END_CASE
END_METHOD

// Alternative to Load. Only works with SINT or BYTE. Result is copied to output.
METHOD PUBLIC LoadToByte : BYTE
VAR_INPUT
	in	: BYTE;			// Set or reset a bit in this integer
	val	: BOOL;			// The value to set
	N	: USINT(0..7);	// position of bit on the nth position from right (right is lowest bit)
END_VAR

// This is a separate method from Load(), because ANY_INT cannot be a reference.
LoadToByte	:= TO_BYTE(Util.PUTBIT(
						X	:= in,
						N	:= N,
						B	:= val));
END_METHOD

// Alternative to Load. Only works with DINT or DWORD. Result is copied to output.
METHOD PUBLIC LoadToDWord : DWORD
VAR_INPUT
	in	: DWORD;		// Set or reset a bit in this integer
	val	: BOOL;			// The value to set
	N	: USINT(0..31);	// position of bit on the nth position from right (right is lowest bit)
END_VAR

// This is a separate method from Load(), because ANY_INT cannot be a reference.
LoadToDWord	:= Util.PUTBIT(
						X	:= in,
						N	:= N,
						B	:= val);
END_METHOD

// Alternative to Load. Only works with INT or WORD. Result is copied to output.
METHOD PUBLIC LoadToWord : WORD
VAR_INPUT
	in	: WORD;			// Set or reset a bit in this integer
	val	: BOOL;			// The value to set
	N	: USINT(0..15);	// position of bit on the nth position from right (right is lowest bit)
END_VAR

// This is a separate method from Load(), because ANY_INT cannot be a reference.
LoadToWord	:= TO_WORD(Util.PUTBIT(
						X	:= in,
						N	:= N,
						B	:= val));
END_METHOD

// Toggles a bit in any integer at position N
METHOD PUBLIC Toggle
VAR_INPUT
	in	: ANY_INT;		// extract bit from this integer
	N	: USINT(0..63);	// position of bit on the nth position from right (right is lowest bit)
END_VAR
ValidateInput(in.diSize, N);

uInput.p1_Byte := in.pValue;

CASE in.diSize OF
	1:	uInput.p1_Byte^		:= SHL( BYTE#1, N) XOR in.pValue^;
	2:	uInput.p2_Word^		:= SHL( WORD#1, N) XOR in.pValue^;
	4:	uInput.p4_DWord^	:= SHL(DWORD#1, N) XOR in.pValue^;
	8:	uInput.p8_LWord^	:= SHL(LWORD#1, N) XOR in.pValue^;
END_CASE
END_METHOD

METHOD PRIVATE ValidateInput
VAR_INPUT
	diSize	: DINT;
	N		: USINT;
END_VAR
IF diSize = 1 AND N > 7
OR diSize = 2 AND N > 15
OR diSize = 4 AND N > 31
THEN
	ThrowException('Invalid parameter; index too large');
END_IF
END_METHOD

(* ---- ClearProducts.prg ---- *)
// Helper functions to clear product (or stack) data
{attribute 'no_explicit_call' := 'Static helper class with methods to reset product data'}
{attribute 'hide_all_locals'}
PROGRAM ClearProducts
VAR
	upper, lower, i, j		: DINT;
END_VAR
VAR CONSTANT
	// Empty product struct that we use to override and initialize product data
	emptyProduct			: ProductType		:= (Present := FALSE);
	emptyStack				: StackStatusType	:= (Present := FALSE, Initialized := TRUE);
END_VAR

END_PROGRAM

// Clear an array of products
METHOD PUBLIC Array1D
VAR_IN_OUT
	aProducts			: ARRAY[*] OF ProductType;
END_VAR
lower	:= LOWER_BOUND(aProducts, 1);
upper	:= UPPER_BOUND(aProducts, 1);

FOR i := lower TO upper DO
	Single(aProducts[i]);
END_FOR
END_METHOD

// Clear a two-dimensional array of products
METHOD PUBLIC Array2D
VAR_IN_OUT
	aProducts			: ARRAY[*,*] OF ProductType;
END_VAR
lower	:= LOWER_BOUND(aProducts, 1);
upper	:= UPPER_BOUND(aProducts, 1);

FOR i := lower TO upper DO
	FOR j := LOWER_BOUND(aProducts, 2) TO UPPER_BOUND(aProducts, 2) DO
		Single(aProducts[i, j]);
	END_FOR
END_FOR
END_METHOD

// Clear all products in a (stack) mould
METHOD PUBLIC Mould
VAR_IN_OUT
	aProducts			: ARRAY[1..GVL_Constants.MaxMouldLevels] OF ARRAY[1..GVL_Constants.MaxProductsInX, 1..GVL_Constants.MaxProductsInY] OF ProductType;
END_VAR
VAR
	k					: DINT;
END_VAR
FOR k := 1 TO GVL_Constants.MaxMouldLevels DO
	Array2D(aProducts[k]);
END_FOR
END_METHOD

// Clear all data in a Product struct
METHOD PUBLIC Single
VAR_IN_OUT
	Product				: ProductType;
END_VAR
Product	:= emptyProduct;
END_METHOD

// Clear all data in a Stack struct
METHOD PUBLIC Stack
VAR_INPUT
	clearStack			: REFERENCE TO StackStatusType;
END_VAR
IF __ISVALIDREF(clearStack) THEN
	clearStack	:= emptyStack;
END_IF
END_METHOD

// Clear an array of stacks
METHOD PUBLIC StackArray1D
VAR_IN_OUT
	aStacks			: ARRAY[*] OF StackStatusType;
END_VAR
lower	:= LOWER_BOUND(aStacks, 1);
upper	:= UPPER_BOUND(aStacks, 1);

FOR i := lower TO upper DO
	Stack(aStacks[i]);
END_FOR
END_METHOD

// Clear a two-dimensional array of stacks
METHOD PUBLIC StackArray2D
VAR_IN_OUT
	aStacks			: ARRAY[*,*] OF StackStatusType;
END_VAR
lower	:= LOWER_BOUND(aStacks, 1);
upper	:= UPPER_BOUND(aStacks, 1);

FOR i := lower TO upper DO
	FOR j := LOWER_BOUND(aStacks, 2) TO UPPER_BOUND(aStacks, 2) DO
		Stack(aStacks[i, j]);
	END_FOR
END_FOR
END_METHOD

(* ---- Increment.prg ---- *)
// Helper functions to increment numbers
{attribute 'no_explicit_call' := 'Static helper class to do simple increment on any number'}
{attribute 'hide_all_locals'}
PROGRAM Increment
VAR
	uInput		: PointerSizesUnion;
END_VAR

END_PROGRAM

// Increment any integer with x when a condition is true
METHOD PUBLIC AnyInt
VAR_INPUT
	input		: ANY_INT;				// Number to increment
	incrementBy	: INT		:= 1;		// Input increments with this value (optional; defaults to 1)
	condition	: BOOL		:= TRUE;	// Only increment when the condition is true (optional)
END_VAR
IF NOT condition THEN
	RETURN;
END_IF

uInput.p1_Byte := input.pValue;

CASE input.diSize OF
	1:	uInput.p1_Sint^	:= uInput.p1_Sint^	+ TO_SINT(incrementBy);
	2:	uInput.p2_Int^	:= uInput.p2_Int^	+ incrementBy;
	4:	uInput.p4_Dint^	:= uInput.p4_Dint^	+ incrementBy;
	8:	uInput.p8_Lint^	:= uInput.p8_Lint^	+ incrementBy;
END_CASE
END_METHOD

// Increment any floating point with x when a condition is true
METHOD PUBLIC AnyReal
VAR_INPUT
	input		: ANY_REAL;				// Number to increment
	incrementBy	: REAL		:= 1.0;		// Input increments with this value (optional; defaults to 1)
	condition	: BOOL		:= TRUE;	// Only increment when the condition is true (optional)
END_VAR
IF NOT condition THEN
	RETURN;
END_IF

uInput.p1_Byte := input.pValue;

CASE input.diSize OF
	4:	uInput.p4_Real^		:= uInput.p4_Real^	+ incrementBy;
	8:	uInput.p8_LReal^	:= uInput.p8_LReal^	+ incrementBy;
END_CASE
END_METHOD

// Increment any integer with x when a condition is true, rollover to Zero when larger than a maximum
METHOD PUBLIC Rollover
VAR_INPUT
	input		: ANY_INT;				// Number to increment
	rollover	: INT;					// When Input larger than this, reset input to zeroValue (endpoint is inclusive)
	incrementBy	: INT		:= 1;		// Input increments with this value (optional; defaults to 1)
	zeroValue	: INT		:= 0;		// Input resets to this value (optional; defaults to 0)
	condition	: BOOL		:= TRUE;	// Only increment when the condition is true (optional)
END_VAR
IF NOT condition THEN
	RETURN;
END_IF

uInput.p1_Byte := input.pValue;

CASE input.diSize OF
	1:	uInput.p1_Sint^	:= TO_SINT(	SEL(uInput.p1_Sint^	+ incrementBy > rollover, uInput.p1_Sint^	+ incrementBy, zeroValue));
	2:	uInput.p2_Int^	:=			SEL(uInput.p2_Int^	+ incrementBy > rollover, uInput.p2_Int^	+ incrementBy, zeroValue);
	4:	uInput.p4_Dint^	:=			SEL(uInput.p4_Dint^	+ incrementBy > rollover, uInput.p4_Dint^	+ incrementBy, zeroValue);
	8:	uInput.p8_Lint^	:=			SEL(uInput.p8_Lint^	+ incrementBy > rollover, uInput.p8_Lint^	+ incrementBy, zeroValue);
END_CASE

// Example; Call function with these parameters:
//
// iState := 0;
// FOR i := 1 TO 999 DO
//	Increment.Rollover(iState, 5, 1, 2);
// END_FOR
//
// iState will be:
// 1, 2, 3, 4, 5, 2, 3, 4, 5, 2, 3, etc.
END_METHOD

// Await the result of a boolean condition and then change the state to a new state
METHOD PUBLIC State
VAR_INPUT
	input		: ANY_INT;				// Number to increment
	condition	: BOOL;					// Only increment when the condition is true
	newState	: DINT;
END_VAR
IF NOT condition THEN
	RETURN;
END_IF

uInput.p1_Byte := input.pValue;

CASE input.diSize OF
	1:	uInput.p1_Sint^	:= TO_SINT(newState);
	2:	uInput.p2_Int^	:= TO_INT(newState);
	4:	uInput.p4_Dint^	:= newState;
	8:	uInput.p8_Lint^	:= newState;
END_CASE
END_METHOD

// Await the result of a enum condition and then change the state to a new state
METHOD PUBLIC StateEnum
VAR_INPUT
	input		: ANY_INT;				// Number to increment
	condition	: enumResultGeneric;	// Only increment when there is a result
	newSuccessState	: DINT;
	newErrorState	: DINT;
END_VAR
IF condition = enumResultGeneric.NoResult THEN
	RETURN;
END_IF

uInput.p1_Byte := input.pValue;

CASE input.diSize OF
	1:	uInput.p1_Sint^	:= TO_SINT(	SEL(condition = enumResultGeneric.Success, newErrorState, newSuccessState));
	2:	uInput.p2_Int^	:= TO_INT(	SEL(condition = enumResultGeneric.Success, newErrorState, newSuccessState));
	4:	uInput.p4_Dint^	:=			SEL(condition = enumResultGeneric.Success, newErrorState, newSuccessState);
	8:	uInput.p8_Lint^	:=			SEL(condition = enumResultGeneric.Success, newErrorState, newSuccessState);
END_CASE
END_METHOD

// Increment any subrange number with x when a condition is true, rollover to lower_limit when larger than upper_limit
METHOD PUBLIC Subrange
VAR_INPUT
	input		: ANY;					// Subrange number to increment (for example INT(4..6)
	lower_limit	: INT;					// Lower limit of the subrange type
	upper_limit : INT;					// Upper limit of the subrange type
	incrementBy	: INT		:= 1;		// Input increments with this value (optional; defaults to 1)
	condition	: BOOL		:= TRUE;	// Only increment when the condition is true (optional)
END_VAR

// (Method is needed because subrange type numbers are not part of ANY_INT. That is why we need input of type ANY)
IF input.TypeClass <> TYPE_CLASS.TYPE_SUBRANGE THEN
	RETURN;
END_IF

IF NOT condition THEN
	RETURN;
END_IF

uInput.p1_Byte := input.pValue;

CASE input.diSize OF
	1:	uInput.p1_Sint^	:= TO_SINT(	SEL(uInput.p1_Sint^	+ incrementBy > upper_limit, uInput.p1_Sint^	+ incrementBy, lower_limit));
	2:	uInput.p2_Int^	:=			SEL(uInput.p2_Int^	+ incrementBy > upper_limit, uInput.p2_Int^		+ incrementBy, lower_limit);
	4:	uInput.p4_Dint^	:=			SEL(uInput.p4_Dint^	+ incrementBy > upper_limit, uInput.p4_Dint^	+ incrementBy, lower_limit);
	8:	uInput.p8_Lint^	:=			SEL(uInput.p8_Lint^	+ incrementBy > upper_limit, uInput.p8_Lint^	+ incrementBy, lower_limit);
END_CASE
END_METHOD

(* ---- LogPlc.prg ---- *)
// Helper functions to log messages to the PLC log
{attribute 'no_explicit_call' := 'Static helper class to log different messages to the PLC log'}
{attribute 'hide_all_locals'}
PROGRAM LogPlc
VAR
	throwFatalMessages		: BOOL;
END_VAR

END_PROGRAM

// Only log when a global option is enabled.
METHOD PUBLIC Debug
VAR_INPUT
	message : STRING(80);
END_VAR
IF GlobalVars.EnableDebugLogging THEN
	LogPlc.Info(message);
END_IF
END_METHOD

METHOD PUBLIC Error
VAR_INPUT
	message : STRING(80);
END_VAR
L_LA.L_AddLog2(
	eSeverity		:= L_TSeverity.L_LogError,	// Severity = 'Trouble log'
	udiComponendID	:= 16#3F03,		// Component ID, reserved range 0x2800 .... 0x3fff
	sLogPayLoad		:= message,
	dwErrorID		:= 0,
	strLanguageTable:= '');
END_METHOD

METHOD PUBLIC Fatal
VAR_INPUT
	message : STRING(80);
END_VAR
L_LA.L_AddLog2(
	eSeverity		:= L_TSeverity.L_LogFatalError,
	udiComponendID	:= 16#3F04,		// Component ID, reserved range 0x2800 .... 0x3fff
	sLogPayLoad		:= message,
	dwErrorID		:= 0,
	strLanguageTable:= '');

IF throwFatalMessages THEN
	Throw();
END_IF
END_METHOD

METHOD PUBLIC Info
VAR_INPUT
	message : STRING(80);
END_VAR
L_LA.L_AddLog2(
	eSeverity		:= L_TSeverity.L_LogInformation,
	udiComponendID	:= 16#3F01,		// Component ID, reserved range 0x2800 .... 0x3fff
	sLogPayLoad		:= message,
	dwErrorID		:= 0,
	strLanguageTable:= '');
END_METHOD

METHOD INTERNAL Throw
VAR
	pApp			: POINTER TO CmpApp.APPLICATION;
	iecResult		: SysTypes.RTS_IEC_RESULT;
END_VAR
// Get handle to current PLC application
pApp := CmpApp.AppGetCurrent(pResult := ADR(iecResult));
IF pApp <> 0 THEN
	// Throw exception in current app
	CmpApp.AppGenerateException(pApp := pApp, ulException := 16#10);	// Throw exception of type: RtsExceptions.RTSEXCPT_WATCHDOG
END_IF

// Note: RTSEXCPT_WATCHDOG exceptions are the only type still working in C5x0 PLCs!
// Other types of exceptions are not working. The PLC does not stop.
// See email from Lenze on 2024-08-20
END_METHOD

METHOD PUBLIC Warn
VAR_INPUT
	message : STRING(80);
END_VAR
L_LA.L_AddLog2(
	eSeverity		:= L_TSeverity.L_LogWarning,
	udiComponendID	:= 16#3F02,		// Component ID, reserved range 0x2800 .... 0x3fff
	sLogPayLoad		:= message,
	dwErrorID		:= 0,
	strLanguageTable:= '');
END_METHOD

(* ---- ModuloTools.prg ---- *)
// Helper functions for module axes
{attribute 'no_explicit_call' := 'Static helper class for modulo functions'}
{attribute 'hide_all_locals'}
PROGRAM ModuloTools
VAR
END_VAR

END_PROGRAM

// Calculate distance of a product on a chain. Rollover is corrected.
METHOD PUBLIC GetDistance : REAL
VAR_INPUT
	productPos		: REAL;		// Position of product on conveyor or chain (mm)
	rollover		: LREAL;	// Rollover (mm)
	actPos			: REAL;		// Current position (mm)
END_VAR
VAR
	delta			: REAL;
END_VAR
// Difference of the 2 positions is how far the product has moved on the conveyor
delta		:= actPos - productPos;

// Correct distance for the rollover
GetDistance	:= SetPosition(delta, rollover);
END_METHOD

// Check if a position lies within a window. Rollover is corrected.
METHOD PUBLIC PositionInWindow : BOOL
VAR_INPUT
	position		: REAL;			// Position to check
	rollover		: LREAL;		// Rollover (mm)
	windowMin		: REAL;			// Position must be >= windowMin
	windowMax		: REAL;			// Position must be <= windowMax
END_VAR

(* Use like this to check camera position on chain:
result := ModuloTools.PositionInWindow(
			position	:= actPos,
			rollover	:= CycleLength,
			windowMin	:= ModuloTools.SetPosition(
								setPos		:= targetPos - adjustTriggerPosition,
								rollover	:= CycleLength),
			windowMax	:= ModuloTools.SetPosition(
								setPos		:= targetPos + 1,
								rollover	:= CycleLength));
*)
// There is no rollover in the window
IF windowMin <= windowMax THEN
	PositionInWindow	:= position >= windowMin AND position <= windowMax;

// Position to check is in the first half of the module cycle length
ELSIF position < TO_REAL(rollover) / 2 THEN
	PositionInWindow	:= position < windowMax;

ELSE
	PositionInWindow	:= position > windowMin;
END_IF
END_METHOD

// Check if position is on a step somewhere on the chain
METHOD PUBLIC PositionOnStep : BOOL
VAR_INPUT
	position		: REAL;			// Position to check
	stepDistance	: REAL;
	hysteresis		: REAL	:= 1;	// Max allowed difference
END_VAR
VAR
	delta			: REAL;
END_VAR
// Get the remainder of position / stepDistance. This is how much the position is different.
delta := TO_REAL( TO_DINT(position * 10) MOD TO_DINT(stepDistance * 10) ) / 10;

// Delta goes from 0 to stepDistance. Change this so it is the shortest distance to a step.
delta := SEL(	delta < stepDistance - delta,
				stepDistance - delta,
				delta);

// delta goes from - half-stepDistance to + half-stepDistance

PositionOnStep := delta <= hysteresis;
END_METHOD

// Check if position is on a step with offset somewhere on the chain.
// Use this to check a sensor on a chain during movement.
METHOD PUBLIC PositionOnStepWithOffset : BOOL
VAR_INPUT
	position		: REAL;			// Position to check
	stepDistance	: REAL;
	hysteresisStart	: REAL;			// Max allowed difference
	hysteresisEnd	: REAL;			// Max allowed difference
END_VAR
VAR
	delta			: REAL;
END_VAR

(* Example how to use:
rejectSensorValid	:= Data.rejectSensorOffset = 0
				OR_ELSE ModuloTools.PositionOnStepWithOffset(
							position		:= Drive.rActPosition,
							stepDistance	:= Data.Step.rPos,
							hysteresisStart	:= Data.rejectSensorOffset[1],
							hysteresisEnd	:= Data.rejectSensorOffset[1] + 10);

alarmActive			:= rejectSensorValid AND NOT sensorRowIsEmpty;
*)
// Get the remainder of position / stepDistance. This is how much the position is different.
delta := TO_REAL( TO_DINT(position * 10) MOD TO_DINT(stepDistance * 10) ) / 10;

// Delta goes from 0 to stepDistance.

PositionOnStepWithOffset := PositionInWindow(
								position		:= delta,
								rollover		:= stepDistance,
								windowMin		:= SetPosition(
														position	:= hysteresisStart,
														rollOver	:= stepDistance),
								windowMax		:= SetPosition(
														position	:= hysteresisEnd,
														rollOver	:= stepDistance),);
END_METHOD

// Check if two positions match for a Modulo axis (within rHysteresis mm).
METHOD PUBLIC PositionReached : BOOL
VAR_INPUT
	actPos			: REAL;			// Actual encoder position
	setPos			: REAL;			// Set position of drive
	rollover		: LREAL;		// Rollover (mm)
	hysteresis		: REAL	:= 1;	// Max allowed difference
END_VAR
PositionReached	:= PositionInWindow(
						actPos,
						rollover,
						SetPosition(setPos - hysteresis, rollover),
						SetPosition(setPos + hysteresis, rollover));
END_METHOD

// Make sure that the set position is always between 0 and rollover.
METHOD PUBLIC SetPosition : REAL
VAR_INPUT
	position		: REAL;			// Position where to move the chain to
	rollover		: LREAL;		// Rollover (mm)
END_VAR
VAR
	correctedPos	: REAL;
END_VAR
IF rollover < 0.001 THEN	// Exception happens when rollover is zero
	SetPosition		:= 0.0;
	RETURN;
END_IF

correctedPos		:= position;

WHILE correctedPos > TO_REAL(rollover) DO
	correctedPos	:= correctedPos - TO_REAL(rollover);
END_WHILE

WHILE correctedPos < 0.0 DO
	correctedPos	:= correctedPos + TO_REAL(rollover);
END_WHILE

SetPosition			:= correctedPos;
END_METHOD
